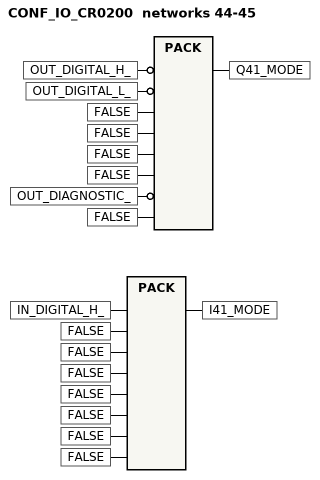
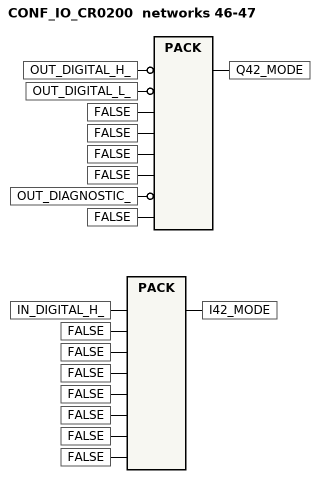
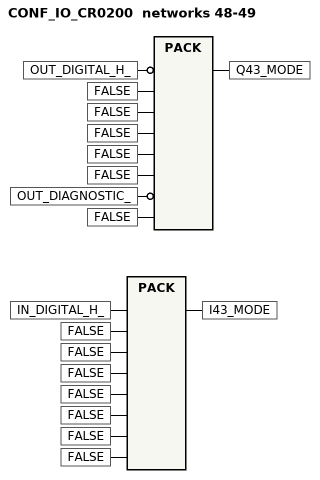
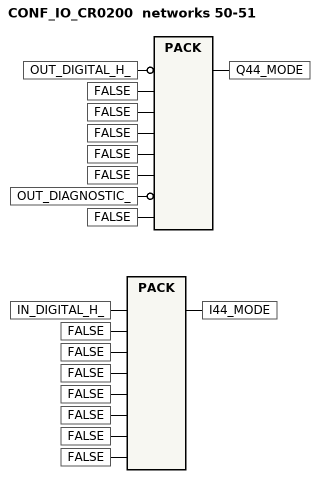
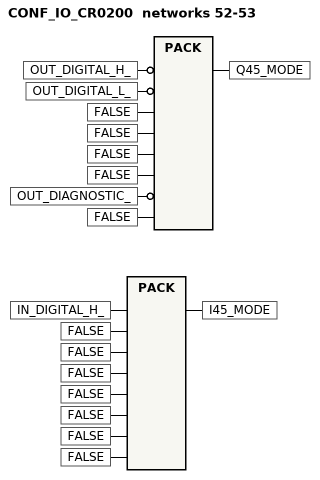
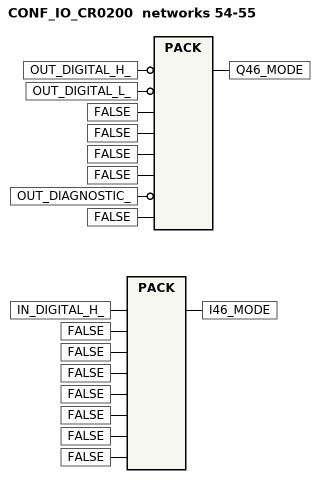
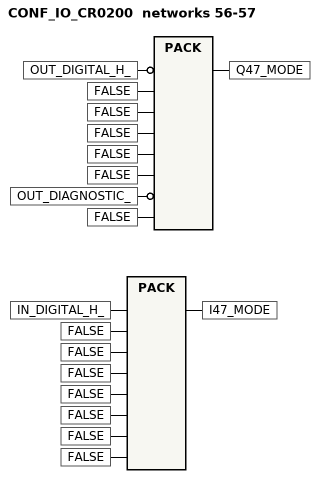
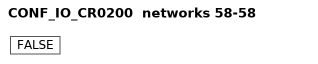
_FBD_ (* Function Block Diagram *)
NETWORK 1
	NOT INIT => >>END
NETWORK 2 (* Configuration byte for analog channel 0 pin 08 Connector 1. No output is connected to this pin. / Default setting:B0:=TRUE,B1:= FALSE,B2:= FALSE,B3:= FALSE,B4:= TRUE,B5:= FALSE,B6:= FALSE,B7:=FALSE *)
	PACK(IN_DIGITAL_H_, FALSE, NOT IN_CURRENT_, NOT IN_VOLTAGE10_, IN_VOLTAGE30_, NOT IN_RATIO_, FALSE, FALSE) => I00_MODE
NETWORK 3 (* Configuration byte for analog channel 1 pin 27 Connector 1. No output is connected to this pin. / Default setting:B0:=TRUE,B1:= FALSE,B2:= FALSE,B3:= FALSE,B4:= TRUE,B5:= FALSE,B6:= FALSE,B7:=FALSE *)
	PACK(IN_DIGITAL_H_, FALSE, NOT IN_CURRENT_, NOT IN_VOLTAGE10_, IN_VOLTAGE30_, NOT IN_RATIO_, FALSE, FALSE) => I01_MODE
NETWORK 4 (* Configuration byte for analog channel 2 pin 09 Connector 1. No output is connected to this pin. / Default setting:B0:=TRUE,B1:= FALSE,B2:= FALSE,B3:= FALSE,B4:= TRUE,B5:= FALSE,B6:= FALSE,B7:=FALSE *)
	PACK(IN_DIGITAL_H_, FALSE, NOT IN_CURRENT_, NOT IN_VOLTAGE10_, IN_VOLTAGE30_, NOT IN_RATIO_, FALSE, FALSE) => I02_MODE
NETWORK 5 (* Configuration byte for analog channel 3 pin 28 Connector 1. No output is connected to this pin. / Default setting:B0:=TRUE,B1:= FALSE,B2:= FALSE,B3:= FALSE,B4:= TRUE,B5:= FALSE,B6:= FALSE,B7:=FALSE *)
	PACK(IN_DIGITAL_H_, FALSE, NOT IN_CURRENT_, NOT IN_VOLTAGE10_, IN_VOLTAGE30_, NOT IN_RATIO_, FALSE, FALSE) => I03_MODE
NETWORK 6 (* Configuration byte for analog channel 4 pin 10 Connector 1. No output is connected to this pin. / Default setting:B0:=TRUE,B1:= FALSE,B2:= FALSE,B3:= FALSE,B4:= TRUE,B5:= FALSE,B6:= FALSE,B7:=FALSE *)
	PACK(IN_DIGITAL_H_, FALSE, NOT IN_CURRENT_, NOT IN_VOLTAGE10_, IN_VOLTAGE30_, NOT IN_RATIO_, FALSE, FALSE) => I04_MODE
NETWORK 7 (* Configuration byte for analog channel 5 pin 29 Connector 1. No output is connected to this pin. / Default setting:B0:=TRUE,B1:= FALSE,B2:= FALSE,B3:= FALSE,B4:= TRUE,B5:= FALSE,B6:= FALSE,B7:=FALSE *)
	PACK(IN_DIGITAL_H_, FALSE, NOT IN_CURRENT_, NOT IN_VOLTAGE10_, IN_VOLTAGE30_, NOT IN_RATIO_, FALSE, FALSE) => I05_MODE
NETWORK 8 (* Configuration byte for analog channel 6 pin 11 Connector 1. No output is connected to this pin. / Default setting:B0:=TRUE,B1:= FALSE,B2:= FALSE,B3:= FALSE,B4:= TRUE,B5:= FALSE,B6:= FALSE,B7:=FALSE *)
	PACK(IN_DIGITAL_H_, FALSE, NOT IN_CURRENT_, NOT IN_VOLTAGE10_, IN_VOLTAGE30_, NOT IN_RATIO_, FALSE, FALSE) => I06_MODE
NETWORK 9 (* Configuration byte for analog channel 7 pin 30 Connector 1. No output is connected to this pin. / Default setting:B0:=TRUE,B1:= FALSE,B2:= FALSE,B3:= FALSE,B4:= TRUE,B5:= FALSE,B6:= FALSE,B7:=FALSE *)
	PACK(IN_DIGITAL_H_, FALSE, NOT IN_CURRENT_, NOT IN_VOLTAGE10_, IN_VOLTAGE30_, NOT IN_RATIO_, FALSE, FALSE) => I07_MODE
NETWORK 10 (* Configuration byte for input %IX0.12  pin 20 Connector 1. No output is connected to this pin. / Default setting:B0:=TRUE,B1:= FALSE,B2:= FALSE,B3:= FALSE,B4:= FALSE,B5:= FALSE,B6:= FALSE,B7:=FALSE *)
	PACK(IN_DIGITAL_H_, FALSE, FALSE, FALSE, FALSE, FALSE, FALSE, NOT IN_FAST_) => I14_MODE
NETWORK 11 (* Configuration byte for input %IX0.13  pin 02 Connector 1. No output is connected to this pin. / Default setting:B0:=TRUE,B1:= FALSE,B2:= FALSE,B3:= FALSE,B4:= FALSE,B5:= FALSE,B6:= FALSE,B7:=FALSE *)
	PACK(IN_DIGITAL_H_, FALSE, FALSE, FALSE, FALSE, FALSE, FALSE, NOT IN_FAST_) => I15_MODE
NETWORK 12 (* Configuration byte for input %IX0.14  pin 21 Connector 1. No output is connected to this pin. / Default setting:B0:=TRUE,B1:= FALSE,B2:= FALSE,B3:= FALSE,B4:= FALSE,B5:= FALSE,B6:= FALSE,B7:=FALSE *)
	PACK(IN_DIGITAL_H_, FALSE, FALSE, FALSE, FALSE, FALSE, FALSE, NOT IN_FAST_) => I16_MODE
NETWORK 13 (* Configuration byte for input %IX0.15  pin 38 Connector 1. No output is connected to this pin. / Default setting:B0:=TRUE,B1:= FALSE,B2:= FALSE,B3:= FALSE,B4:= FALSE,B5:= FALSE,B6:= FALSE,B7:=FALSE *)
	PACK(IN_DIGITAL_H_, FALSE, FALSE, FALSE, FALSE, FALSE, FALSE, NOT IN_FAST_) => I17_MODE
NETWORK 14 (* Configuration byte for input %IX1.04  pin 19 Connector 1. No output is connected to this pin. / Default setting:B0:=TRUE,B1:= FALSE,B2:= FALSE,B3:= FALSE,B4:= FALSE,B5:= FALSE,B6:= FALSE,B7:=FALSE *)
	PACK(IN_DIGITAL_H_, FALSE, FALSE, FALSE, FALSE, FALSE, FALSE, NOT IN_FAST_) => I24_MODE
NETWORK 15 (* Configuration byte for input %IX1.05  pin 55 Connector 1. No output is connected to this pin. / Default setting:B0:=TRUE,B1:= FALSE,B2:= FALSE,B3:= FALSE,B4:= FALSE,B5:= FALSE,B6:= FALSE,B7:=FALSE *)
	PACK(IN_DIGITAL_H_, FALSE, FALSE, FALSE, FALSE, FALSE, FALSE, NOT IN_FAST_) => I25_MODE
NETWORK 16 (* Configuration byte for input %IX1.06  pin 18 Connector 1. No output is connected to this pin. / Default setting:B0:=TRUE,B1:= FALSE,B2:= FALSE,B3:= FALSE,B4:= FALSE,B5:= FALSE,B6:= FALSE,B7:=FALSE *)
	PACK(IN_DIGITAL_H_, FALSE, FALSE, FALSE, FALSE, FALSE, FALSE, NOT IN_FAST_) => I26_MODE
NETWORK 17 (* Configuration byte for input %IX1.07  pin 37 Connector 1. No output is connected to this pin. / Default setting:B0:=TRUE,B1:= FALSE,B2:= FALSE,B3:= FALSE,B4:= FALSE,B5:= FALSE,B6:= FALSE,B7:=FALSE *)
	PACK(IN_DIGITAL_H_, FALSE, FALSE, FALSE, FALSE, FALSE, FALSE, NOT IN_FAST_) => I27_MODE
NETWORK 18 (* Configuration byte for output %QX0.00  pin 44 Connector 1. The input %IX0.08 on pin 44 has no configuration byte. / Default setting:B0:=TRUE,B1:= FALSE,B2:= FALSE,B3:= FALSE,B4:= FALSE,B5:= FALSE,B6:= FALSE,B7:=TRUE *)
	PACK(OUT_DIGITAL_H_, FALSE, NOT OUT_CURRENT_, FALSE, FALSE, FALSE, NOT OUT_DIAGNOSTIC_, OUT_OVERLOAD_PROTECTION_) => Q10_MODE
NETWORK 19 (* Configuration byte for output %QX0.01  pin 45 Connector 1. The input %IX0.09 on pin 45 has no configuration byte. / Default setting:B0:=TRUE,B1:= FALSE,B2:= FALSE,B3:= FALSE,B4:= FALSE,B5:= FALSE,B6:= FALSE,B7:=TRUE *)
	PACK(OUT_DIGITAL_H_, FALSE, NOT OUT_CURRENT_, FALSE, FALSE, FALSE, NOT OUT_DIAGNOSTIC_, OUT_OVERLOAD_PROTECTION_) => Q11_MODE
NETWORK 20 (* Configuration byte for output %QX0.02  pin 46 Connector 1. The input %IX0.10 on pin 46 has no configuration byte. / Default setting:B0:=TRUE,B1:= FALSE,B2:= FALSE,B3:= FALSE,B4:= FALSE,B5:= FALSE,B6:= FALSE,B7:=TRUE *)
	PACK(OUT_DIGITAL_H_, FALSE, NOT OUT_CURRENT_, FALSE, FALSE, FALSE, NOT OUT_DIAGNOSTIC_, OUT_OVERLOAD_PROTECTION_) => Q12_MODE
NETWORK 21 (* Configuration byte for output %QX0.03  pin 47 Connector 1. The input %IX0.11 on pin 47 has no configuration byte. / Default setting:B0:=TRUE,B1:= FALSE,B2:= FALSE,B3:= FALSE,B4:= FALSE,B5:= FALSE,B6:= FALSE,B7:=TRUE *)
	PACK(OUT_DIGITAL_H_, FALSE, NOT OUT_CURRENT_, FALSE, FALSE, FALSE, NOT OUT_DIAGNOSTIC_, OUT_OVERLOAD_PROTECTION_) => Q13_MODE
NETWORK 22 (* Configuration byte for output %QX0.04  pin 36 Connector 1. The input %IX1.00 on pin 36 has no configuration byte. / Default setting:B0:=TRUE,B1:= FALSE,B2:= FALSE,B3:= FALSE,B4:= FALSE,B5:= FALSE,B6:= FALSE,B7:=TRUE *)
	PACK(OUT_DIGITAL_H_, FALSE, NOT OUT_CURRENT_, FALSE, FALSE, FALSE, NOT OUT_DIAGNOSTIC_, OUT_OVERLOAD_PROTECTION_) => Q20_MODE
NETWORK 23 (* Configuration byte for output %QX0.05  pin 54 Connector 1 The input %IX1.01 on pin 54 has no configuration byte. / Default setting:B0:=TRUE,B1:= FALSE,B2:= FALSE,B3:= FALSE,B4:= FALSE,B5:= FALSE,B6:= FALSE,B7:=TRUE *)
	PACK(OUT_DIGITAL_H_, FALSE, NOT OUT_CURRENT_, FALSE, FALSE, FALSE, NOT OUT_DIAGNOSTIC_, OUT_OVERLOAD_PROTECTION_) => Q21_MODE
NETWORK 24 (* Configuration byte for output %QX0.06  pin 17 Connector 1 The input %IX1.02 on pin 17 has no configuration byte. / Default setting:B0:=TRUE,B1:= FALSE,B2:= FALSE,B3:= FALSE,B4:= FALSE,B5:= FALSE,B6:= FALSE,B7:=TRUE *)
	PACK(OUT_DIGITAL_H_, FALSE, NOT OUT_CURRENT_, FALSE, FALSE, FALSE, NOT OUT_DIAGNOSTIC_, OUT_OVERLOAD_PROTECTION_) => Q22_MODE
NETWORK 25 (* Configuration byte for output %QX0.07  pin 53 Connector 1 The input %IX1.03 on pin 53 has no configuration byte. / Default setting:B0:=TRUE,B1:= FALSE,B2:= FALSE,B3:= FALSE,B4:= FALSE,B5:= FALSE,B6:= FALSE,B7:=TRUE *)
	PACK(OUT_DIGITAL_H_, FALSE, NOT OUT_CURRENT_, FALSE, FALSE, FALSE, NOT OUT_DIAGNOSTIC_, OUT_OVERLOAD_PROTECTION_) => Q23_MODE
NETWORK 26 (* Configuration byte for output %QX0.08  pin 39 Connector 1. / Default setting:B0:=TRUE,B1:= FALSE,B2:= FALSE,B3:= FALSE,B4:= FALSE,B5:= FALSE,B6:= FALSE,B7:=FALSE *)
	PACK(OUT_DIGITAL_H_, FALSE, FALSE, FALSE, FALSE, FALSE, NOT OUT_DIAGNOSTIC_, FALSE) => Q30_MODE
NETWORK 27 (* Configuration byte for input %IX1.08  pin 39 Connector 1. / Default setting:B0:=TRUE,B1:= FALSE,B2:= FALSE,B3:= FALSE,B4:= FALSE,B5:= FALSE,B6:= FALSE,B7:=FALSE *)
	PACK(IN_DIGITAL_H_, NOT IN_DIGITAL_L_, FALSE, FALSE, FALSE, FALSE, FALSE, FALSE) => I30_MODE
NETWORK 28 (* Configuration byte for output %QX0.09  pin 03 Connector 1. / Default setting:B0:=TRUE,B1:= FALSE,B2:= FALSE,B3:= FALSE,B4:= FALSE,B5:= FALSE,B6:= FALSE,B7:=FALSE *)
	PACK(OUT_DIGITAL_H_, FALSE, FALSE, FALSE, FALSE, FALSE, NOT OUT_DIAGNOSTIC_, FALSE) => Q31_MODE
NETWORK 29 (* Configuration byte for input %IX1.09  pin 03 Connector 1. / Default setting:B0:=TRUE,B1:= FALSE,B2:= FALSE,B3:= FALSE,B4:= FALSE,B5:= FALSE,B6:= FALSE,B7:=FALSE *)
	PACK(IN_DIGITAL_H_, NOT IN_DIGITAL_L_, FALSE, FALSE, FALSE, FALSE, FALSE, FALSE) => I31_MODE
NETWORK 30 (* Configuration byte for output %QX0.10  pin 40 Connector 1. / Default setting:B0:=TRUE,B1:= FALSE,B2:= FALSE,B3:= FALSE,B4:= FALSE,B5:= FALSE,B6:= FALSE,B7:=FALSE *)
	PACK(OUT_DIGITAL_H_, FALSE, FALSE, FALSE, FALSE, FALSE, NOT OUT_DIAGNOSTIC_, FALSE) => Q32_MODE
NETWORK 31 (* Configuration byte forintput %IX1.10  pin 40 Connector 1. / Default setting:B0:=TRUE,B1:= FALSE,B2:= FALSE,B3:= FALSE,B4:= FALSE,B5:= FALSE,B6:= FALSE,B7:=FALSE *)
	PACK(IN_DIGITAL_H_, NOT IN_DIGITAL_L_, FALSE, FALSE, FALSE, FALSE, FALSE, FALSE) => I32_MODE
NETWORK 32 (* Configuration byte for output %QX0.11  pin 22 Connector 1. / Default setting:B0:=TRUE,B1:= FALSE,B2:= FALSE,B3:= FALSE,B4:= FALSE,B5:= FALSE,B6:= FALSE,B7:=FALSE *)
	PACK(OUT_DIGITAL_H_, FALSE, FALSE, FALSE, FALSE, FALSE, NOT OUT_DIAGNOSTIC_, FALSE) => Q33_MODE
NETWORK 33 (* Configuration byte for input %IX1.11  pin 22 Connector 1. / Default setting:B0:=TRUE,B1:= FALSE,B2:= FALSE,B3:= FALSE,B4:= FALSE,B5:= FALSE,B6:= FALSE,B7:=FALSE *)
	PACK(IN_DIGITAL_H_, NOT IN_DIGITAL_L_, FALSE, FALSE, FALSE, FALSE, FALSE, FALSE) => I33_MODE
NETWORK 34 (* Configuration byte for output %QX0.12  pin 41 Connector 1. / Default setting:B0:=TRUE,B1:= FALSE,B2:= FALSE,B3:= FALSE,B4:= FALSE,B5:= FALSE,B6:= FALSE,B7:=FALSE *)
	PACK(OUT_DIGITAL_H_, FALSE, FALSE, FALSE, FALSE, FALSE, NOT OUT_DIAGNOSTIC_, FALSE) => Q34_MODE
NETWORK 35 (* Configuration byte for input %IX1.12  pin 41 Connector 1. / Default setting:B0:=TRUE,B1:= FALSE,B2:= FALSE,B3:= FALSE,B4:= FALSE,B5:= FALSE,B6:= FALSE,B7:=FALSE *)
	PACK(IN_DIGITAL_H_, NOT IN_DIGITAL_L_, FALSE, FALSE, FALSE, FALSE, FALSE, FALSE) => I34_MODE
NETWORK 36 (* Configuration byte for output %QX0.13  pin 42 Connector 1. / Default setting:B0:=TRUE,B1:= FALSE,B2:= FALSE,B3:= FALSE,B4:= FALSE,B5:= FALSE,B6:= FALSE,B7:=FALSE *)
	PACK(OUT_DIGITAL_H_, FALSE, FALSE, FALSE, FALSE, FALSE, NOT OUT_DIAGNOSTIC_, FALSE) => Q35_MODE
NETWORK 37 (* Configuration byte for input %IX1.13  pin 42 Connector 1. / Default setting:B0:=TRUE,B1:= FALSE,B2:= FALSE,B3:= FALSE,B4:= FALSE,B5:= FALSE,B6:= FALSE,B7:=FALSE *)
	PACK(IN_DIGITAL_H_, NOT IN_DIGITAL_L_, FALSE, FALSE, FALSE, FALSE, FALSE, FALSE) => I35_MODE
NETWORK 38 (* Configuration byte for output %QX0.14  pin 43 Connector 1. / Default setting:B0:=TRUE,B1:= FALSE,B2:= FALSE,B3:= FALSE,B4:= FALSE,B5:= FALSE,B6:= FALSE,B7:=FALSE *)
	PACK(OUT_DIGITAL_H_, FALSE, FALSE, FALSE, FALSE, FALSE, NOT OUT_DIAGNOSTIC_, FALSE) => Q36_MODE
NETWORK 39 (* Configuration byte for input %IX1.14  pin 43 Connector 1. / Default setting:B0:=TRUE,B1:= FALSE,B2:= FALSE,B3:= FALSE,B4:= FALSE,B5:= FALSE,B6:= FALSE,B7:=FALSE *)
	PACK(IN_DIGITAL_H_, NOT IN_DIGITAL_L_, FALSE, FALSE, FALSE, FALSE, FALSE, FALSE) => I36_MODE
NETWORK 40 (* Configuration byte for output %QX0.15  pin 04 Connector 1. / Default setting:B0:=TRUE,B1:= FALSE,B2:= FALSE,B3:= FALSE,B4:= FALSE,B5:= FALSE,B6:= FALSE,B7:=FALSE *)
	PACK(OUT_DIGITAL_H_, FALSE, FALSE, FALSE, FALSE, FALSE, NOT OUT_DIAGNOSTIC_, FALSE) => Q37_MODE
NETWORK 41 (* Configuration byte for input %IX1.15  pin 04 Connector 1. / Default setting:B0:=TRUE,B1:= FALSE,B2:= FALSE,B3:= FALSE,B4:= FALSE,B5:= FALSE,B6:= FALSE,B7:=FALSE *)
	PACK(IN_DIGITAL_H_, NOT IN_DIGITAL_L_, FALSE, FALSE, FALSE, FALSE, FALSE, FALSE) => I37_MODE
NETWORK 42 (* Configuration byte for output %QX1.00  pin 48 Connector 1. / Default setting:B0:=FALSE,B1:= FALSE,B2:= FALSE,B3:= FALSE,B4:= FALSE,B5:= FALSE,B6:= FALSE,B7:=FALSE *)
	PACK(NOT OUT_DIGITAL_H_, FALSE, FALSE, FALSE, FALSE, FALSE, NOT OUT_DIAGNOSTIC_, FALSE) => Q40_MODE
NETWORK 43 (* Configuration byte for intput %IX2.00  pin 48 Connector 1. / Default setting:B0:=TRUE,B1:= FALSE,B2:= FALSE,B3:= FALSE,B4:= FALSE,B5:= FALSE,B6:= FALSE,B7:=FALSE *)
	PACK(IN_DIGITAL_H_, FALSE, FALSE, FALSE, FALSE, FALSE, FALSE, FALSE) => I40_MODE
NETWORK 44 (* Configuration byte for output %QX1.01  pin 49 Connector 1. / Default setting:B0:=FALSE,B1:= FALSE,B2:= FALSE,B3:= FALSE,B4:= FALSE,B5:= FALSE,B6:= FALSE,B7:=FALSE *)
	PACK(NOT OUT_DIGITAL_H_, NOT OUT_DIGITAL_L_, FALSE, FALSE, FALSE, FALSE, NOT OUT_DIAGNOSTIC_, FALSE) => Q41_MODE
NETWORK 45 (* Configuration byte for input %IX2.01  pin 49 Connector 1. / Default setting:B0:=TRUE,B1:= FALSE,B2:= FALSE,B3:= FALSE,B4:= FALSE,B5:= FALSE,B6:= FALSE,B7:=FALSE *)
	PACK(IN_DIGITAL_H_, FALSE, FALSE, FALSE, FALSE, FALSE, FALSE, FALSE) => I41_MODE
NETWORK 46 (* Configuration byte for output %QX1.02  pin 31 Connector 1. / Default setting:B0:=FALSE,B1:= FALSE,B2:= FALSE,B3:= FALSE,B4:= FALSE,B5:= FALSE,B6:= FALSE,B7:=FALSE *)
	PACK(NOT OUT_DIGITAL_H_, NOT OUT_DIGITAL_L_, FALSE, FALSE, FALSE, FALSE, NOT OUT_DIAGNOSTIC_, FALSE) => Q42_MODE
NETWORK 47 (* Configuration byte for input %IX2.02  pin 31 Connector 1. / Default setting:B0:=TRUE,B1:= FALSE,B2:= FALSE,B3:= FALSE,B4:= FALSE,B5:= FALSE,B6:= FALSE,B7:=FALSE *)
	PACK(IN_DIGITAL_H_, FALSE, FALSE, FALSE, FALSE, FALSE, FALSE, FALSE) => I42_MODE
NETWORK 48 (* Configuration byte for output %QX1.03  pin 50 Connector 1. / Default setting:B0:=FALSE,B1:= FALSE,B2:= FALSE,B3:= FALSE,B4:= FALSE,B5:= FALSE,B6:= FALSE,B7:=FALSE *)
	PACK(NOT OUT_DIGITAL_H_, FALSE, FALSE, FALSE, FALSE, FALSE, NOT OUT_DIAGNOSTIC_, FALSE) => Q43_MODE
NETWORK 49 (* Configuration byte for input %IX2.03  pin 50 Connector 1. / Default setting:B0:=TRUE,B1:= FALSE,B2:= FALSE,B3:= FALSE,B4:= FALSE,B5:= FALSE,B6:= FALSE,B7:=FALSE *)
	PACK(IN_DIGITAL_H_, FALSE, FALSE, FALSE, FALSE, FALSE, FALSE, FALSE) => I43_MODE
NETWORK 50 (* Configuration byte for output %QX1.04  pin 51 Connector 1. / Default setting:B0:=FALSE,B1:= FALSE,B2:= FALSE,B3:= FALSE,B4:= FALSE,B5:= FALSE,B6:= FALSE,B7:=FALSE *)
	PACK(NOT OUT_DIGITAL_H_, FALSE, FALSE, FALSE, FALSE, FALSE, NOT OUT_DIAGNOSTIC_, FALSE) => Q44_MODE
NETWORK 51 (* Configuration byte for input %IX2.04  pin 51 Connector 1. / Default setting:B0:=TRUE,B1:= FALSE,B2:= FALSE,B3:= FALSE,B4:= FALSE,B5:= FALSE,B6:= FALSE,B7:=FALSE *)
	PACK(IN_DIGITAL_H_, FALSE, FALSE, FALSE, FALSE, FALSE, FALSE, FALSE) => I44_MODE
NETWORK 52 (* Configuration byte for output %QX1.05  pin 52 Connector 1. / Default setting:B0:=FALSE,B1:= FALSE,B2:= FALSE,B3:= FALSE,B4:= FALSE,B5:= FALSE,B6:= FALSE,B7:=FALSE *)
	PACK(NOT OUT_DIGITAL_H_, NOT OUT_DIGITAL_L_, FALSE, FALSE, FALSE, FALSE, NOT OUT_DIAGNOSTIC_, FALSE) => Q45_MODE
NETWORK 53 (* Configuration byte for input %IX1.05  pin 52 Connector 1. / Default setting:B0:=TRUE,B1:= FALSE,B2:= FALSE,B3:= FALSE,B4:= FALSE,B5:= FALSE,B6:= FALSE,B7:=FALSE *)
	PACK(IN_DIGITAL_H_, FALSE, FALSE, FALSE, FALSE, FALSE, FALSE, FALSE) => I45_MODE
NETWORK 54 (* Configuration byte for output %QX1.06  pin 16 Connector 1. / Default setting:B0:=FALSE,B1:= FALSE,B2:= FALSE,B3:= FALSE,B4:= FALSE,B5:= FALSE,B6:= FALSE,B7:=FALSE *)
	PACK(NOT OUT_DIGITAL_H_, NOT OUT_DIGITAL_L_, FALSE, FALSE, FALSE, FALSE, NOT OUT_DIAGNOSTIC_, FALSE) => Q46_MODE
NETWORK 55 (* Configuration byte for input %IX2.06  pin 16 Connector 1. / Default setting:B0:=TRUE,B1:= FALSE,B2:= FALSE,B3:= FALSE,B4:= FALSE,B5:= FALSE,B6:= FALSE,B7:=FALSE *)
	PACK(IN_DIGITAL_H_, FALSE, FALSE, FALSE, FALSE, FALSE, FALSE, FALSE) => I46_MODE
NETWORK 56 (* Configuration byte for output %QX1.07  pin 35 Connector 1. / Default setting:B0:=FALSE,B1:= FALSE,B2:= FALSE,B3:= FALSE,B4:= FALSE,B5:= FALSE,B6:= FALSE,B7:=FALSE *)
	PACK(NOT OUT_DIGITAL_H_, FALSE, FALSE, FALSE, FALSE, FALSE, NOT OUT_DIAGNOSTIC_, FALSE) => Q47_MODE
NETWORK 57 (* Configuration byte for input %IX2.07  pin 35 Connector 1. / Default setting:B0:=TRUE,B1:= FALSE,B2:= FALSE,B3:= FALSE,B4:= FALSE,B5:= FALSE,B6:= FALSE,B7:=FALSE *)
	PACK(IN_DIGITAL_H_, FALSE, FALSE, FALSE, FALSE, FALSE, FALSE, FALSE) => I47_MODE
NETWORK 58 END::
	FALSE
_END_FBD_
END_PROGRAM

(* POU I_O_CONFIGURATION/CONF_IO_CR0200_E, FBD *)
PROGRAM CONF_IO_CR0200_E
VAR

END_VAR
VAR CONSTANT

	(*IN_NOMODE ==> all Bits 0*)
	IN_DIGITAL_H_ : BOOL := TRUE;	(*Bit 0*)
	IN_DIGITAL_L_ : BOOL:= TRUE;		(*Bit 1*)
	IN_CURRENT_ : BOOL := TRUE;	(*Bit 2*)
	IN_VOLTAGE10_ : BOOL := TRUE;	(*Bit 3*)
	IN_VOLTAGE30_ : BOOL := TRUE;	(*Bit 4*)
	IN_RATIO_ : BOOL := TRUE;			(*Bit 5*)
	IN_DIAGNOSTIC_ : BOOL := TRUE;	(*Bit 6*)

	IN_FAST_ : BOOL := TRUE;			(*Bit 7 *)

	(*OUT_NOMODE ==> all bits 0*)
	OUT_DIGITAL_H_ : BOOL := TRUE;						(*Bit 0*)
	OUT_DIGITAL_L_ : BOOL := TRUE;						(*Bit 1*)
	OUT_CURRENT_ : BOOL := TRUE;						(*Bit 2*)

	OUT_DIAGNOSTIC_ : BOOL := TRUE;					(*Bit 6*)
	OUT_OVERLOAD_PROTECTION_ : BOOL := TRUE;	(*Bit 7*)

END_VAR

VAR_INPUT
	init: BOOL;
END_VAR
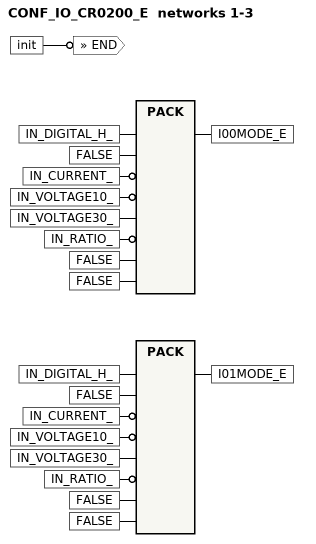
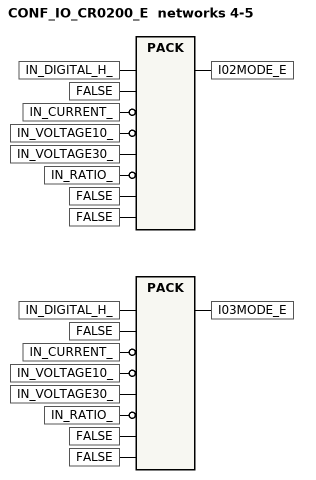
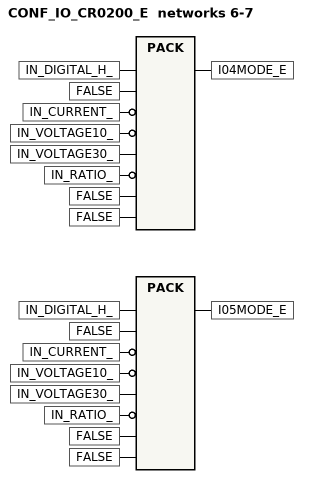
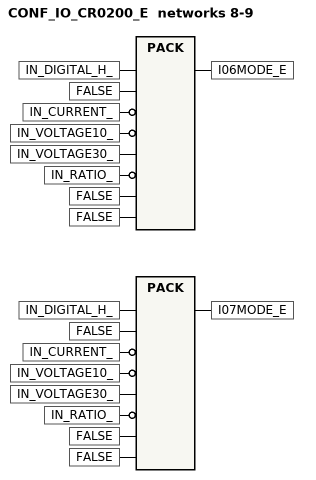
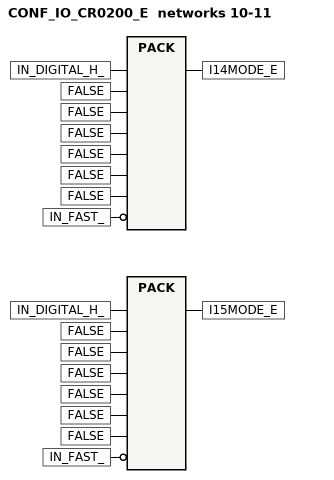
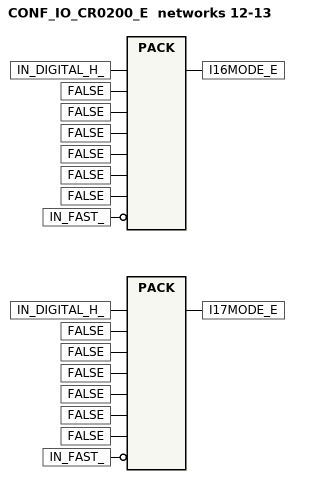
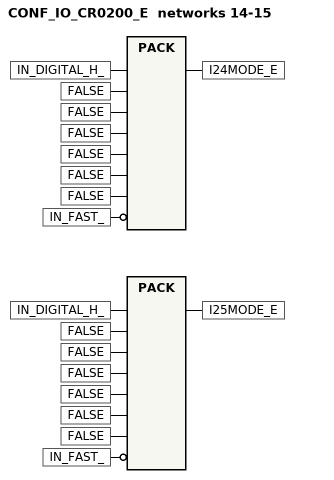
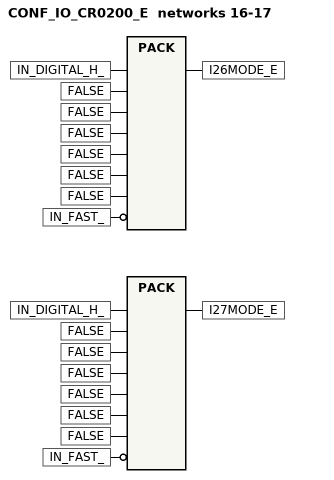
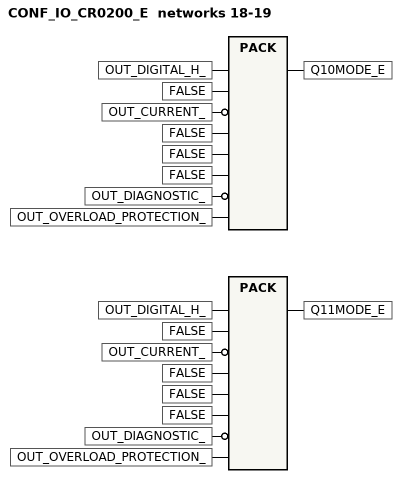
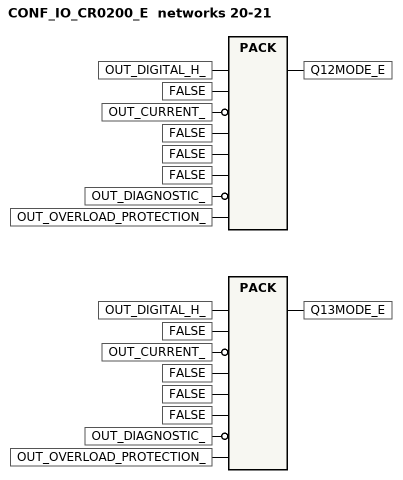
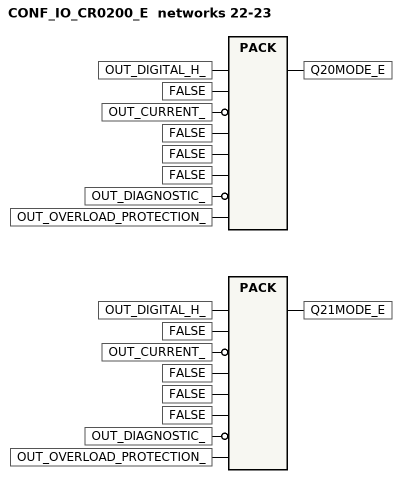
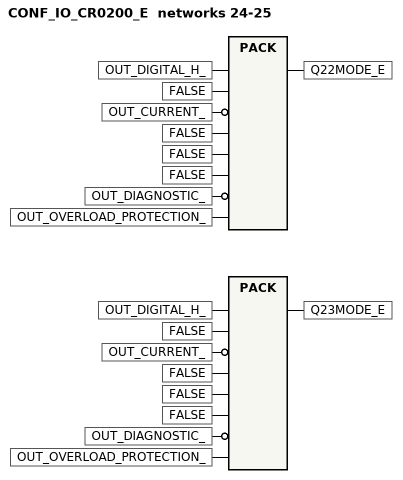
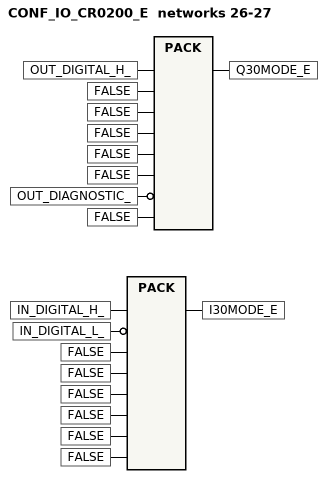
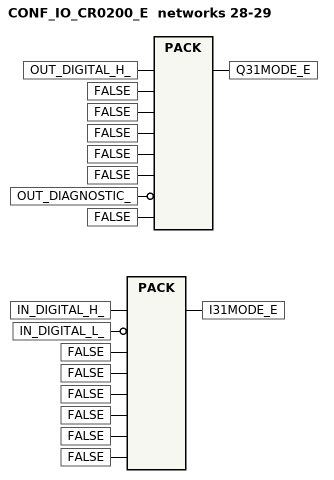
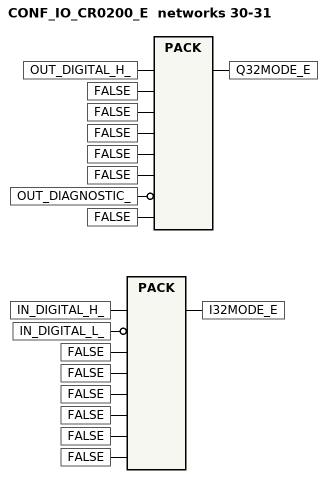
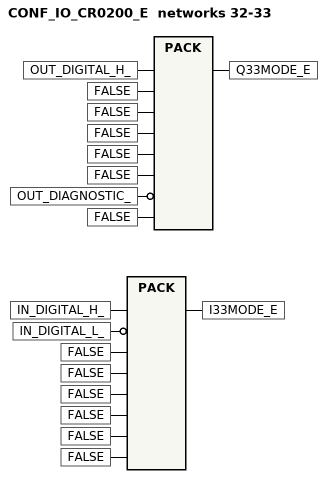
